{attribute 'qualified_only'}
VAR_GLOBAL PERSISTENT
	{attribute 'OPC.UA.DA' := '1'}	
	// Indicates if object creating and deleting counted in ObjectStatistics
	CountObjectStatistics : BOOL;
END_VAR

(* stored: Version 1.1.0.1
   GVL ObjectStatisticsSettings: Id {7f924c5f-0383-4dfc-a181-e3d9714446b9} *)
